// TIA Portal V17 export
// export: Created 2024-08-07T21:43:57.5148333Z, ExportSetting WithDefaults, DisplayName Totally Integrated Automation Portal, DisplayVersion V17 Update 7, DisplayName TIA Portal Openness, DisplayVersion V17 Update 7, DisplayName TIA Portal Version Control Interface, DisplayVersion V17, DisplayName SINAMICS Startdrive Advanced, DisplayVersion V17 SP2, DisplayName SINAMICS Startdrive G110M, G120, G120C, G120D, G120P, G115D, DisplayVersion V17 SP2, DisplayName SINAMICS Startdrive G130, G150, S120, S150, SINAMICS MV, S210, DisplayVersion V17 SP2, DisplayName STEP 7 Professional, DisplayVersion V17 Update 7, DisplayName STEP 7 Safety, DisplayVersion V17 Update 6, DisplayName WinCC Advanced / Unified PC, DisplayVersion V17 Update 7
FUNCTION_BLOCK "RivetingCycle"   // FB52, LAD
{ S7_Optimized_Access := 'TRUE' }
VERSION : 0.1
// stored: AutoNumber true, IsIECCheckEnabled false, IsRetainMemResEnabled false, MemoryReserve 100, SetENOAutomatically false, UDAEnableTagReadback false
   VAR_INPUT
      parameters : Array[0..2] of USInt;
      basicPosition : Bool;
      twoRivets : Bool;
   END_VAR
   VAR_OUTPUT
      MeasuredData1 { ExternalAccessible := 'False'; ExternalVisible := 'False'; ExternalWritable := 'False'} : "UDT_Friedrich";
      MeasuredData2 { ExternalAccessible := 'False'; ExternalVisible := 'False'; ExternalWritable := 'False'} : "UDT_Friedrich";
   END_VAR
   VAR_IN_OUT
      riveter : "UDT_Friedrich";
      data : "UDT_FittingStatus";
      cylinderSupport : "UDT_Cylinder";
      cylinderShift : "UDT_Cylinder";
   END_VAR
   VAR
      cnt : Int;
      R_TRIG_Instance { S7_SetPoint := 'True'} : R_TRIG;
      IEC_Timer_timeout { S7_SetPoint := 'True'} : TON_TIME;
      R_TRIG_Instance_1 { S7_SetPoint := 'True'} : R_TRIG;
      ton_WayWithTimeoutReached { S7_SetPoint := 'True'} : TON_TIME;
   END_VAR
   VAR_TEMP   // added for the SCL form of the ladder/FBD networks
      _w1 : Bool;
      _w2 : Bool;
   END_VAR
BEGIN

REGION Network 1: Reset cycle
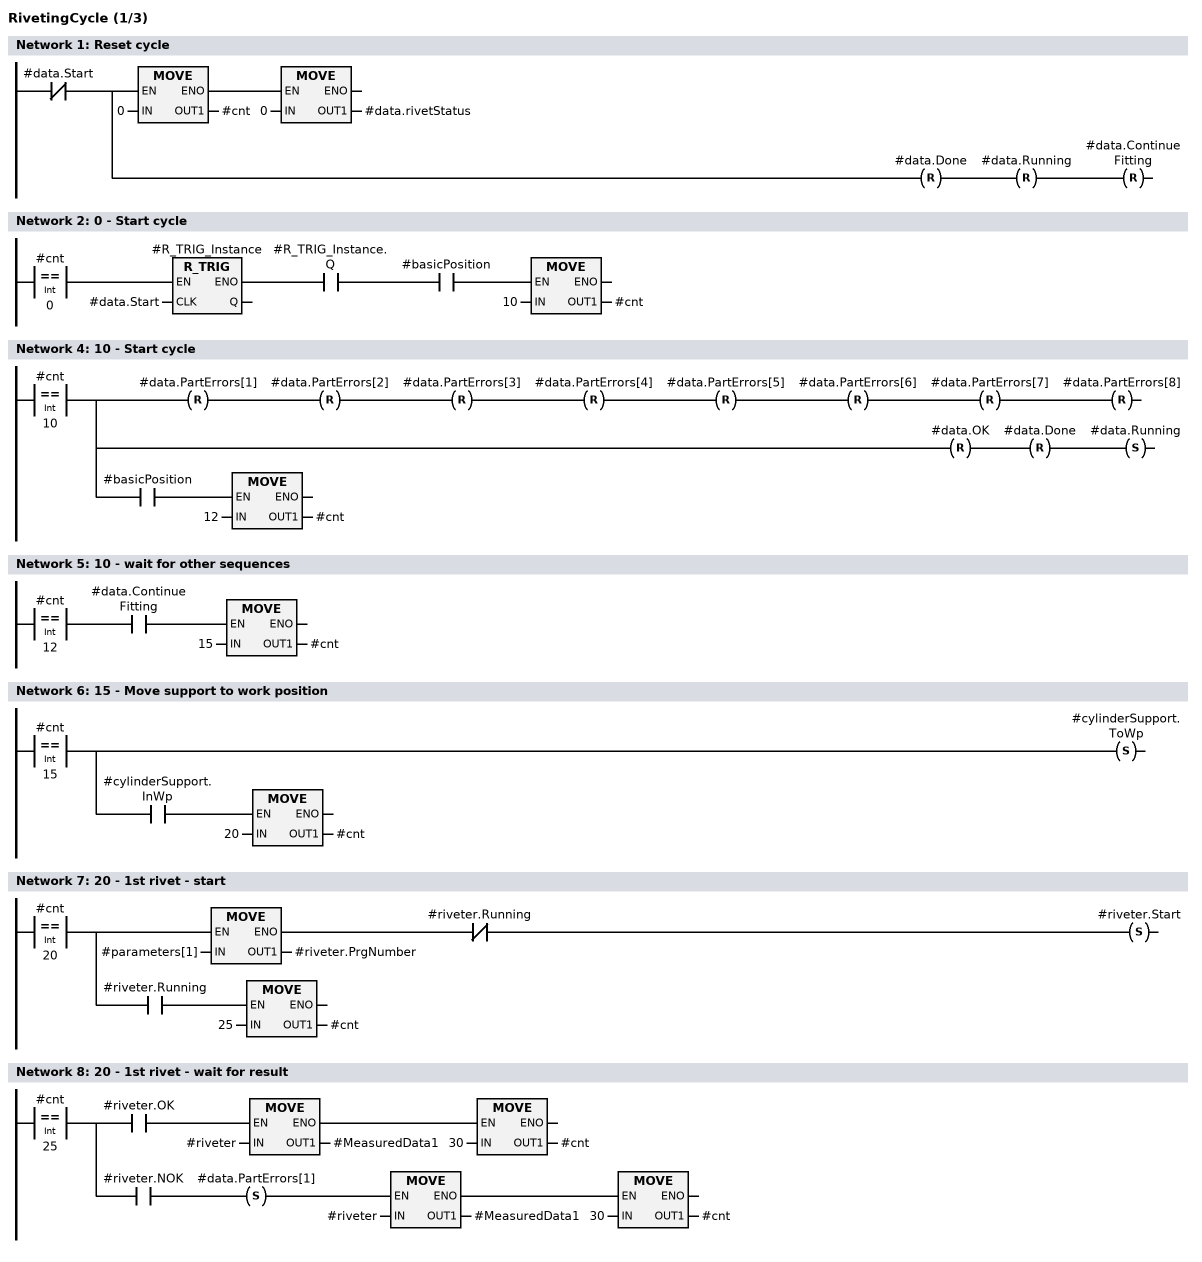
   RUNG wire#powerrail
      I_Contact( #data.Start )
      wire#w1
      Move(in := 0, out1 => #cnt)
      Move(in := 0, out1 => #data.rivetStatus)
   END_RUNG
   RUNG wire#w1
      R_Coil( #data.Done )
      R_Coil( #data.Running )
      R_Coil( #data.ContinueFitting )
   END_RUNG
   // the same network as SCL:
   IF NOT #data.Start THEN
       #cnt := 0;
       #data.rivetStatus := 0;
       #data.Done := FALSE;
       #data.Running := FALSE;
       #data.ContinueFitting := FALSE;
   END_IF;
END_REGION

REGION Network 2: 0 - Start cycle
   RUNG wire#powerrail
      { S7_Templates := "SrcType := Int" } EQ_Contact(in1 := #cnt, in2 := 0)
      #R_TRIG_Instance.R_TRIG(CLK := #data.Start, Q =>)
      Contact( #R_TRIG_Instance.Q )
      Contact( #basicPosition )
      Move(in := 10, out1 => #cnt)
   END_RUNG
   // the same network as SCL:
   #_w1 := #cnt = 0;
   #R_TRIG_Instance(EN := #_w1, CLK := #data.Start, ENO => #_w2);   // R_TRIG
   IF #_w2 AND #R_TRIG_Instance.Q AND #basicPosition THEN #cnt := 10; END_IF;
END_REGION

REGION Network 3 (SCL): 10 - Start cycle - init measured data
   IF #cnt = 10 THEN
       #MeasuredData1.Start := FALSE;
       #MeasuredData1.PrgNumber := 0;
       #MeasuredData1.Ready := FALSE;
       #MeasuredData1.Running := FALSE;
       #MeasuredData1.OK := FALSE;
       #MeasuredData1.NOK := FALSE;
       #MeasuredData1.H1OK := FALSE;
       #MeasuredData1.H2OK := FALSE;
       #MeasuredData1.TimeOK := FALSE;
       #MeasuredData1.StartError := FALSE;
       #MeasuredData1.LastH1 := 0.0;
       #MeasuredData1.LastH2 := 0.0;
       #MeasuredData1.LastTime := 0.0;
       #MeasuredData1.LastZ1 := 0.0;
       #MeasuredData1.Error := FALSE;
       #MeasuredData1.Z1OK := FALSE;
       #MeasuredData1.NewDataAfterStart := FALSE;
       #MeasuredData2 := #MeasuredData1;
   END_IF;
END_REGION

REGION Network 4: 10 - Start cycle
   RUNG wire#powerrail
      { S7_Templates := "SrcType := Int" } EQ_Contact(in1 := #cnt, in2 := 10)
      wire#w1
      R_Coil( #data.PartErrors[1] )
      R_Coil( #data.PartErrors[2] )
      R_Coil( #data.PartErrors[3] )
      R_Coil( #data.PartErrors[4] )
      R_Coil( #data.PartErrors[5] )
      R_Coil( #data.PartErrors[6] )
      R_Coil( #data.PartErrors[7] )
      R_Coil( #data.PartErrors[8] )
   END_RUNG
   RUNG wire#w1
      R_Coil( #data.OK )
      R_Coil( #data.Done )
      S_Coil( #data.Running )
   END_RUNG
   RUNG wire#w1
      Contact( #basicPosition )
      Move(in := 12, out1 => #cnt)
   END_RUNG
   // the same network as SCL:
   #_w1 := #cnt = 10;
   IF #_w1 THEN
       #data.PartErrors[1] := FALSE;
       #data.PartErrors[2] := FALSE;
       #data.PartErrors[3] := FALSE;
       #data.PartErrors[4] := FALSE;
       #data.PartErrors[5] := FALSE;
       #data.PartErrors[6] := FALSE;
       #data.PartErrors[7] := FALSE;
       #data.PartErrors[8] := FALSE;
       #data.OK := FALSE;
       #data.Done := FALSE;
       #data.Running := TRUE;
   END_IF;
   IF #_w1 AND #basicPosition THEN #cnt := 12; END_IF;
END_REGION

REGION Network 5: 10 - wait for other sequences
   RUNG wire#powerrail
      { S7_Templates := "SrcType := Int" } EQ_Contact(in1 := #cnt, in2 := 12)
      Contact( #data.ContinueFitting )
      Move(in := 15, out1 => #cnt)
   END_RUNG
   // the same network as SCL:
   IF (#cnt = 12) AND #data.ContinueFitting THEN #cnt := 15; END_IF;
END_REGION

REGION Network 6: 15 - Move support to work position
   RUNG wire#powerrail
      { S7_Templates := "SrcType := Int" } EQ_Contact(in1 := #cnt, in2 := 15)
      wire#w1
      S_Coil( #cylinderSupport.ToWp )
   END_RUNG
   RUNG wire#w1
      Contact( #cylinderSupport.InWp )
      Move(in := 20, out1 => #cnt)
   END_RUNG
   // the same network as SCL:
   #_w1 := #cnt = 15;
   IF #_w1 THEN #cylinderSupport.ToWp := TRUE; END_IF;
   IF #_w1 AND #cylinderSupport.InWp THEN #cnt := 20; END_IF;
END_REGION

REGION Network 7: 20 - 1st rivet - start
   RUNG wire#powerrail
      { S7_Templates := "SrcType := Int" } EQ_Contact(in1 := #cnt, in2 := 20)
      wire#w1
      Move(in := #parameters[1], out1 => #riveter.PrgNumber)
      I_Contact( #riveter.Running )
      S_Coil( #riveter.Start )
   END_RUNG
   RUNG wire#w1
      Contact( #riveter.Running )
      Move(in := 25, out1 => #cnt)
   END_RUNG
   // the same network as SCL:
   #_w1 := #cnt = 20;
   IF #_w1 THEN #riveter.PrgNumber := #parameters[1]; END_IF;
   IF #_w1 AND NOT #riveter.Running THEN #riveter.Start := TRUE; END_IF;
   IF #_w1 AND #riveter.Running THEN #cnt := 25; END_IF;
END_REGION

REGION Network 8: 20 - 1st rivet - wait for result
   RUNG wire#powerrail
      { S7_Templates := "SrcType := Int" } EQ_Contact(in1 := #cnt, in2 := 25)
      wire#w1
      Contact( #riveter.OK )
      Move(in := #riveter, out1 => #MeasuredData1)
      Move(in := 30, out1 => #cnt)
   END_RUNG
   RUNG wire#w1
      Contact( #riveter.NOK )
      S_Coil( #data.PartErrors[1] )
      Move(in := #riveter, out1 => #MeasuredData1)
      Move(in := 30, out1 => #cnt)
   END_RUNG
   // the same network as SCL:
   #_w1 := #cnt = 25;
   IF #_w1 AND #riveter.OK THEN
       #MeasuredData1 := #riveter;
       #cnt := 30;
   END_IF;
   IF #_w1 AND #riveter.NOK THEN
       #data.PartErrors[1] := TRUE;
       #MeasuredData1 := #riveter;
       #cnt := 30;
   END_IF;
END_REGION

REGION Network 9: 30 - Move support to base position
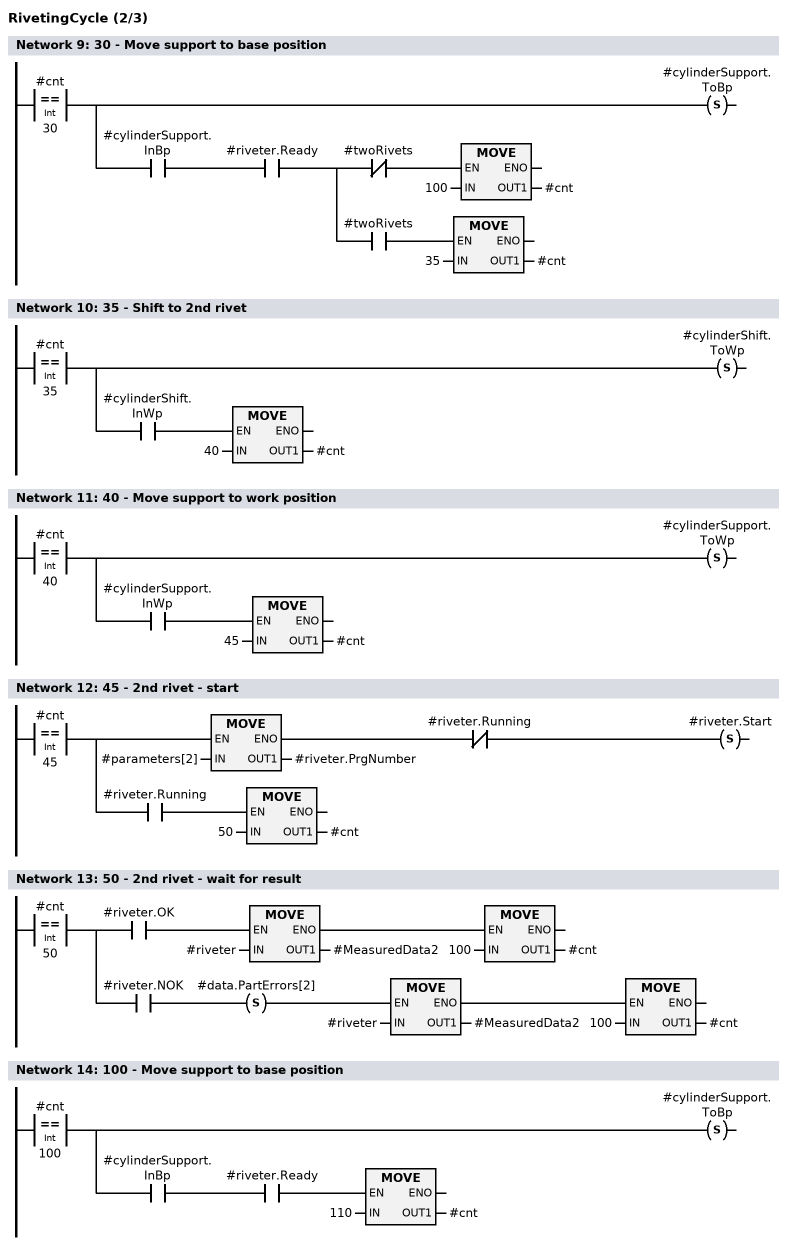
   RUNG wire#powerrail
      { S7_Templates := "SrcType := Int" } EQ_Contact(in1 := #cnt, in2 := 30)
      wire#w1
      S_Coil( #cylinderSupport.ToBp )
   END_RUNG
   RUNG wire#w1
      Contact( #cylinderSupport.InBp )
      Contact( #riveter.Ready )
      wire#w2
      I_Contact( #twoRivets )
      Move(in := 100, out1 => #cnt)
   END_RUNG
   RUNG wire#w2
      Contact( #twoRivets )
      Move(in := 35, out1 => #cnt)
   END_RUNG
   // the same network as SCL:
   #_w1 := #cnt = 30;
   IF #_w1 THEN #cylinderSupport.ToBp := TRUE; END_IF;
   #_w2 := #_w1 AND #cylinderSupport.InBp AND #riveter.Ready;
   IF #_w2 AND NOT #twoRivets THEN #cnt := 100; END_IF;
   IF #_w2 AND #twoRivets THEN #cnt := 35; END_IF;
END_REGION

REGION Network 10: 35 - Shift to 2nd rivet
   RUNG wire#powerrail
      { S7_Templates := "SrcType := Int" } EQ_Contact(in1 := #cnt, in2 := 35)
      wire#w1
      S_Coil( #cylinderShift.ToWp )
   END_RUNG
   RUNG wire#w1
      Contact( #cylinderShift.InWp )
      Move(in := 40, out1 => #cnt)
   END_RUNG
   // the same network as SCL:
   #_w1 := #cnt = 35;
   IF #_w1 THEN #cylinderShift.ToWp := TRUE; END_IF;
   IF #_w1 AND #cylinderShift.InWp THEN #cnt := 40; END_IF;
END_REGION

REGION Network 11: 40 - Move support to work position
   RUNG wire#powerrail
      { S7_Templates := "SrcType := Int" } EQ_Contact(in1 := #cnt, in2 := 40)
      wire#w1
      S_Coil( #cylinderSupport.ToWp )
   END_RUNG
   RUNG wire#w1
      Contact( #cylinderSupport.InWp )
      Move(in := 45, out1 => #cnt)
   END_RUNG
   // the same network as SCL:
   #_w1 := #cnt = 40;
   IF #_w1 THEN #cylinderSupport.ToWp := TRUE; END_IF;
   IF #_w1 AND #cylinderSupport.InWp THEN #cnt := 45; END_IF;
END_REGION

REGION Network 12: 45 - 2nd rivet - start
   RUNG wire#powerrail
      { S7_Templates := "SrcType := Int" } EQ_Contact(in1 := #cnt, in2 := 45)
      wire#w1
      Move(in := #parameters[2], out1 => #riveter.PrgNumber)
      I_Contact( #riveter.Running )
      S_Coil( #riveter.Start )
   END_RUNG
   RUNG wire#w1
      Contact( #riveter.Running )
      Move(in := 50, out1 => #cnt)
   END_RUNG
   // the same network as SCL:
   #_w1 := #cnt = 45;
   IF #_w1 THEN #riveter.PrgNumber := #parameters[2]; END_IF;
   IF #_w1 AND NOT #riveter.Running THEN #riveter.Start := TRUE; END_IF;
   IF #_w1 AND #riveter.Running THEN #cnt := 50; END_IF;
END_REGION

REGION Network 13: 50 - 2nd rivet - wait for result
   RUNG wire#powerrail
      { S7_Templates := "SrcType := Int" } EQ_Contact(in1 := #cnt, in2 := 50)
      wire#w1
      Contact( #riveter.OK )
      Move(in := #riveter, out1 => #MeasuredData2)
      Move(in := 100, out1 => #cnt)
   END_RUNG
   RUNG wire#w1
      Contact( #riveter.NOK )
      S_Coil( #data.PartErrors[2] )
      Move(in := #riveter, out1 => #MeasuredData2)
      Move(in := 100, out1 => #cnt)
   END_RUNG
   // the same network as SCL:
   #_w1 := #cnt = 50;
   IF #_w1 AND #riveter.OK THEN
       #MeasuredData2 := #riveter;
       #cnt := 100;
   END_IF;
   IF #_w1 AND #riveter.NOK THEN
       #data.PartErrors[2] := TRUE;
       #MeasuredData2 := #riveter;
       #cnt := 100;
   END_IF;
END_REGION

REGION Network 14: 100 - Move support to base position
   RUNG wire#powerrail
      { S7_Templates := "SrcType := Int" } EQ_Contact(in1 := #cnt, in2 := 100)
      wire#w1
      S_Coil( #cylinderSupport.ToBp )
   END_RUNG
   RUNG wire#w1
      Contact( #cylinderSupport.InBp )
      Contact( #riveter.Ready )
      Move(in := 110, out1 => #cnt)
   END_RUNG
   // the same network as SCL:
   #_w1 := #cnt = 100;
   IF #_w1 THEN #cylinderSupport.ToBp := TRUE; END_IF;
   IF #_w1 AND #cylinderSupport.InBp AND #riveter.Ready THEN #cnt := 110; END_IF;
END_REGION

REGION Network 15: 110 - Shift to base position
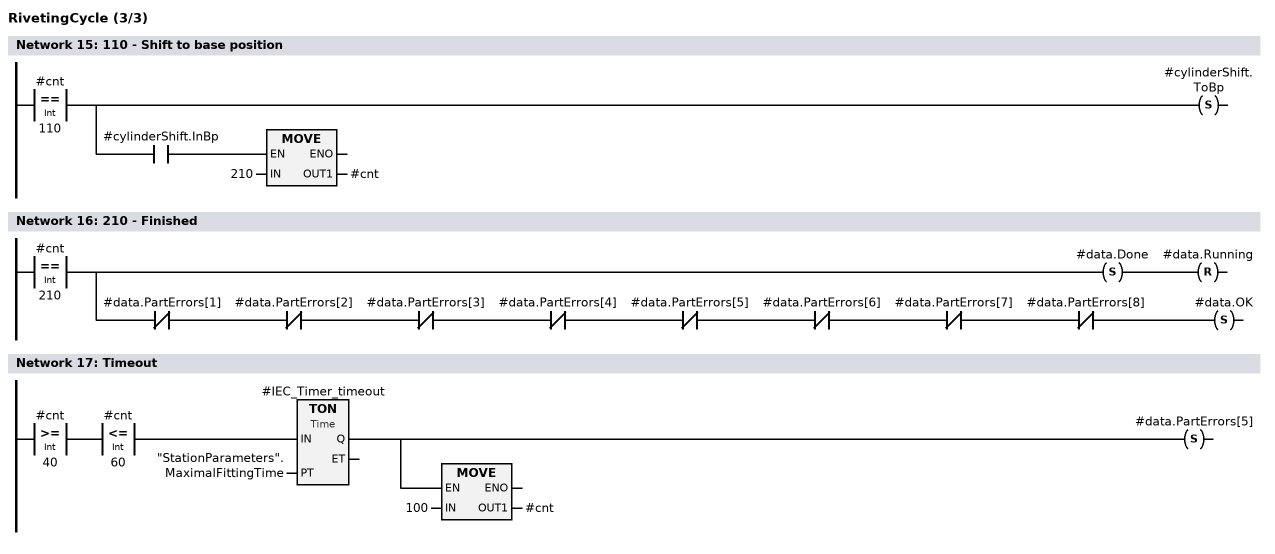
   RUNG wire#powerrail
      { S7_Templates := "SrcType := Int" } EQ_Contact(in1 := #cnt, in2 := 110)
      wire#w1
      S_Coil( #cylinderShift.ToBp )
   END_RUNG
   RUNG wire#w1
      Contact( #cylinderShift.InBp )
      Move(in := 210, out1 => #cnt)
   END_RUNG
   // the same network as SCL:
   #_w1 := #cnt = 110;
   IF #_w1 THEN #cylinderShift.ToBp := TRUE; END_IF;
   IF #_w1 AND #cylinderShift.InBp THEN #cnt := 210; END_IF;
END_REGION

REGION Network 16: 210 - Finished
   RUNG wire#powerrail
      { S7_Templates := "SrcType := Int" } EQ_Contact(in1 := #cnt, in2 := 210)
      wire#w1
      S_Coil( #data.Done )
      R_Coil( #data.Running )
   END_RUNG
   RUNG wire#w1
      I_Contact( #data.PartErrors[1] )
      I_Contact( #data.PartErrors[2] )
      I_Contact( #data.PartErrors[3] )
      I_Contact( #data.PartErrors[4] )
      I_Contact( #data.PartErrors[5] )
      I_Contact( #data.PartErrors[6] )
      I_Contact( #data.PartErrors[7] )
      I_Contact( #data.PartErrors[8] )
      S_Coil( #data.OK )
   END_RUNG
   // the same network as SCL:
   #_w1 := #cnt = 210;
   IF #_w1 THEN
       #data.Done := TRUE;
       #data.Running := FALSE;
   END_IF;
   IF #_w1 AND NOT #data.PartErrors[1] AND NOT #data.PartErrors[2] AND NOT #data.PartErrors[3] AND NOT #data.PartErrors[4] AND NOT #data.PartErrors[5] AND NOT #data.PartErrors[6] AND NOT #data.PartErrors[7] AND NOT #data.PartErrors[8] THEN
       #data.OK := TRUE;
   END_IF;
END_REGION

REGION Network 17: Timeout
   RUNG wire#powerrail
      { S7_Templates := "SrcType := Int" } GE_Contact(in1 := #cnt, in2 := 40)
      { S7_Templates := "SrcType := Int" } LE_Contact(in1 := #cnt, in2 := 60)
      { S7_Templates := "time_type := Time" } #IEC_Timer_timeout.TON(pt := "StationParameters".MaximalFittingTime, et =>)
      wire#w1
      S_Coil( #data.PartErrors[5] )
   END_RUNG
   RUNG wire#w1
      Move(in := 100, out1 => #cnt)
   END_RUNG
   // the same network as SCL:
   #IEC_Timer_timeout(IN := (#cnt >= 40) AND (#cnt <= 60), PT := "StationParameters".MaximalFittingTime);   // TON
   IF #IEC_Timer_timeout.Q THEN
       #data.PartErrors[5] := TRUE;
       #cnt := 100;
   END_IF;
END_REGION
END_FUNCTION_BLOCK
